# B&R Automation Studio project Fertigungsband
Automation Studio 4.9


## Configuration Kamerainspektion

### Task classes (Cpu.sw)
```
Cyclic#4:
  Verpressen <- Verpressen.prg
```


## Configuration Pressen

CPU X20CP1584, AutomationRuntime J4.93, Build 4.1.2, Vc V4.73.2

### Task classes (Cpu.sw)
```
Cyclic#4:
  Verpressen <- Verpressen.prg
Binaries: udbdef, FWRules, TCData, iomap, ashwac, Role, sysconf, arconfig, asfw, User, asiol2, ashwd
```

### Hardware
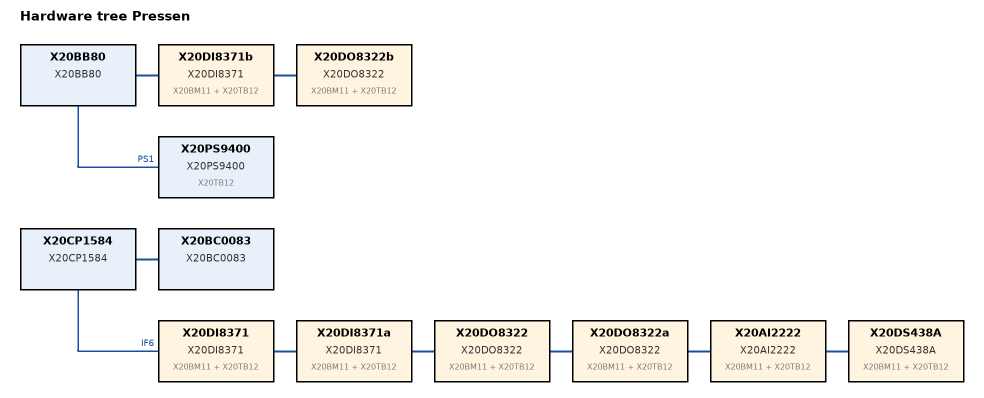
```
X20AI2222 : X20AI2222 v1.2.0.0  [SS1 -> X20TB12d.SS; SL -> X20BM11d.SL1]
X20BB80 : X20BB80 v1.1.0.0
X20BC0083 : X20BC0083 v2.14.0.0  [PLK1 -> X20CP1584.IF3 (NodeNumber=1) [Cable Type=PowerlinkCable, Length=10, Version=1.0.0.3]; SL -> X20BB80.SL1]
X20BM11 : X20BM11 v1.1.0.0  [X2X1 -> X20CP1584.IF6]
X20BM11a : X20BM11 v1.1.0.0  [X2X1 -> X20BM11.X2X2]
X20BM11b : X20BM11 v1.1.0.0  [X2X1 -> X20BM11a.X2X2]
X20BM11c : X20BM11 v1.1.0.0  [X2X1 -> X20BM11b.X2X2]
X20BM11d : X20BM11 v1.1.0.0  [X2X1 -> X20BM11c.X2X2]
X20BM11e : X20BM11 v1.1.0.0  [X2X1 -> X20BM11d.X2X2]
X20BM11f : X20BM11 v1.1.0.0  [X2X1 -> X20BB80.IF1]
X20BM11g : X20BM11 v1.1.0.0  [X2X1 -> X20BM11f.X2X2]
X20CP1584 : X20CP1584 v1.10.0.0
  Connector IF2:
    ActivateDevice = 1
    Mode = Manual
    InternetAddress = 10.36.37.3
    SubnetMask = 255.255.255.0
  ConfigurationID = Fertiungsband_basisConfig
  FileDevice1
  FileDeviceName1 = USER
  FileDevicePath1 = USER_PATH
X20DI8371 : X20DI8371 v1.4.0.0  [SS1 -> X20TB12.SS; SL -> X20BM11.SL1]
X20DI8371a : X20DI8371 v1.4.0.0  [SS1 -> X20TB12a.SS; SL -> X20BM11a.SL1]
X20DI8371b : X20DI8371 v1.4.0.0  [SS1 -> X20TB12g.SS; SL -> X20BM11f.SL1]
X20DO8322 : X20DO8322 v1.5.0.0  [SS1 -> X20TB12b.SS; SL -> X20BM11b.SL1]
X20DO8322a : X20DO8322 v1.5.0.0  [SS1 -> X20TB12c.SS; SL -> X20BM11c.SL1]
X20DO8322b : X20DO8322 v1.5.0.0  [SS1 -> X20TB12h.SS; SL -> X20BM11g.SL1]
X20DS438A : X20DS438A v2.3.0.0  [SS1 -> X20TB12e.SS; SL -> X20BM11e.SL1]
  DtmRef = FBD.BRIOLinkModuleDTM.DTMCore.X20DS438A
  DtmId = 84349467-65e7-4600-9e01-ae0e2285639b
  CommDtmId = 6efde10b-66b8-4cae-87f3-db096a55aaa2
  RequiresDTMBuild = true
  ConfigFile = Communication.dtm
  ConfigModule = asiol2
X20PS9400 : X20PS9400 v1.8.0.0  [SS1 -> X20TB12f.SS; PS -> X20BB80.PS1]
X20TB12 : X20TB12 v1.0.0.0
X20TB12a : X20TB12 v1.0.0.0
X20TB12b : X20TB12 v1.0.0.0
X20TB12c : X20TB12 v1.0.0.0
X20TB12d : X20TB12 v1.0.0.0
X20TB12e : X20TB12 v1.0.0.0
X20TB12f : X20TB12 v1.0.0.0
X20TB12g : X20TB12 v1.0.0.0
X20TB12h : X20TB12 v1.0.0.0
```

### IoMap.iom - X20CP1584/IoMap.iom
```iecst
VAR_CONFIG
	::Werkstueck_Bandende_Links AT %IX."X20DI8371".DigitalInput01;
	::Werkstueck_Bandende_Rechts AT %IX."X20DI8371".DigitalInput02;
	::Koppelsensor_Empfaenger_rechts AT %IX."X20DI8371".DigitalInput03;
	::Koppelsensor_Empfaenger_links AT %IX."X20DI8371".DigitalInput04;
	::Stopper_geoffnet AT %IX."X20DI8371".DigitalInput05;
	::Notaus AT %IX."X20DI8371".DigitalInput06;
	::Motor_Drehgeber1 AT %IX."X20DI8371".DigitalInput07;
	::Motor_Drehgeber2 AT %IX."X20DI8371".DigitalInput08;
	::START_Taster_Gruen AT %IX."X20DI8371a".DigitalInput01;
	::STOP_Taster_Rot AT %IX."X20DI8371a".DigitalInput02;
	::Reset_Taster_Weis AT %IX."X20DI8371a".DigitalInput03;
	::Wahlschalter AT %IX."X20DI8371a".DigitalInput04;
	::AuthCodeBit[0] AT %IX."X20DI8371a".DigitalInput05;
	::AuthCodeBit[1] AT %IX."X20DI8371a".DigitalInput06;
	::AuthCodeBit[2] AT %IX."X20DI8371a".DigitalInput07;
	::AuthCodeBit[3] AT %IX."X20DI8371a".DigitalInput08;
	::Bandantrieb_Rechts AT %QX."X20DO8322".DigitalOutput01;
	::Bandantrieb_Links AT %QX."X20DO8322".DigitalOutput02;
	::Bandantrieb_Schleichgang AT %QX."X20DO8322".DigitalOutput03;
	::Stopper_oeffnen AT %QX."X20DO8322".DigitalOutput04;
	::Koppelsensor_Sender_links AT %QX."X20DO8322".DigitalOutput05;
	::Koppelsensor_Sender_rechts AT %QX."X20DO8322".DigitalOutput06;
	::Lampe_Gruen AT %QX."X20DO8322a".DigitalOutput01;
	::Lampe_Weiss AT %QX."X20DO8322a".DigitalOutput02;
	::Verpressen:Lampe_Q1 AT %QX."X20DO8322a".DigitalOutput03;
	::Verpressen:Lampe_Q2 AT %QX."X20DO8322a".DigitalOutput04;
	::Potentiometer1 AT %IW."X20AI2222".AnalogInput01;
	::Potentiometer2 AT %IW."X20AI2222".AnalogInput02;
	::Verpressen:Zylinder_auf AT %QX."X20DO8322b".DigitalOutput01;
	::Verpressen:Zylinder_ab AT %QX."X20DO8322b".DigitalOutput02;
	::Verpressen:Zylinder_oben AT %IX."X20DI8371b".DigitalInput01;
	::Verpressen:Zylinder_unten AT %IX."X20DI8371b".DigitalInput02;
	::Verpressen:Teil_vorhanden AT %IX."X20DI8371b".DigitalInput08;
END_VAR
```

## Configuration Tunnelofen

### IoMap.iom - X20CP1584/IoMap.iom
```iecst
VAR_CONFIG
	::Werkstueck_Bandende_Links AT %IX."X20DI8371".DigitalInput01;
	::Werkstueck_Bandende_Rechts AT %IX."X20DI8371".DigitalInput02;
	::Koppelsensor_Empfaenger_rechts AT %IX."X20DI8371".DigitalInput03;
	::Koppelsensor_Empfaenger_links AT %IX."X20DI8371".DigitalInput04;
	::Stopper_geoffnet AT %IX."X20DI8371".DigitalInput05;
	::Notaus AT %IX."X20DI8371".DigitalInput06;
	::Motor_Drehgeber1 AT %IX."X20DI8371".DigitalInput07;
	 ::Motor_Drehgeber2 AT %IX."X20DI8371".DigitalInput08;
	::START_Taster_Gruen AT %IX."X20DI8371a".DigitalInput01;
	::STOP_Taster_Rot AT %IX."X20DI8371a".DigitalInput02;
	::Reset_Taster_Weis AT %IX."X20DI8371a".DigitalInput03;
	::Wahlschalter AT %IX."X20DI8371a".DigitalInput04;
	::AuthCodeBit[0] AT %IX."X20DI8371a".DigitalInput05;
	::AuthCodeBit[1] AT %IX."X20DI8371a".DigitalInput06;
	::AuthCodeBit[2]  AT %IX."X20DI8371a".DigitalInput07;
	::AuthCodeBit[3]  AT %IX."X20DI8371a".DigitalInput08;
	::Bandantrieb_Rechts AT %QX."X20DO8322".DigitalOutput01;
	::Bandantrieb_Links AT %QX."X20DO8322".DigitalOutput02;
	::Bandantrieb_Schleichgang AT %QX."X20DO8322".DigitalOutput03;
	::Stopper_oeffnen AT %QX."X20DO8322".DigitalOutput04;
	::Koppelsensor_Sender_links AT %QX."X20DO8322".DigitalOutput05;
	::Koppelsensor_Sender_rechts AT %QX."X20DO8322".DigitalOutput06;
	::Lampe_Gruen AT %QX."X20DO8322a".DigitalOutput01;
	::Lampe_Weiss AT %QX."X20DO8322a".DigitalOutput02;
	::Lampe_Q1_Weiss AT %QX."X20DO8322a".DigitalOutput03;
	::Lampe_Q2_Weiss AT %QX."X20DO8322a".DigitalOutput04;
	::Potentiometer1 AT %IW."X20AI2222".AnalogInput01;
	::Potentiometer2 AT %IW."X20AI2222".AnalogInput02;
END_VAR
```

## Configuration Wenden

CPU X20CP1584, AutomationRuntime J4.93, Build 4.1.2, Vc V4.73.2

### Hardware
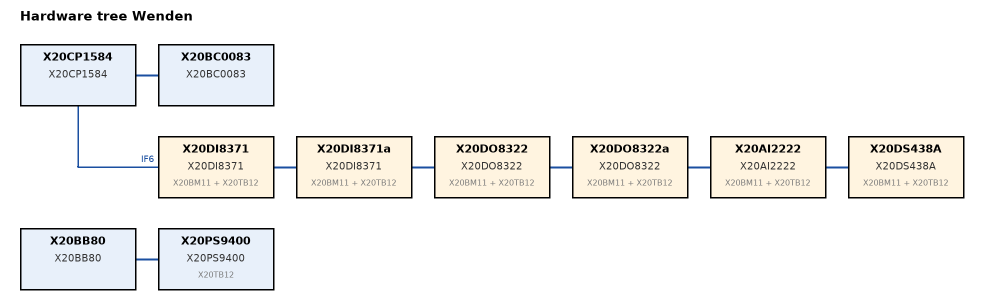
```
X20AI2222 : X20AI2222 v1.2.0.0  [SS1 -> X20TB12d.SS; SL -> X20BM11d.SL1]
X20BB80 : X20BB80 v1.1.0.0
X20BC0083 : X20BC0083 v2.14.0.0  [PLK1 -> X20CP1584.IF3 (NodeNumber=1) [Cable Type=PowerlinkCable, Length=10, Version=1.0.0.3]; SL -> X20BB80.SL1]
X20BM11 : X20BM11 v1.1.0.0  [X2X1 -> X20CP1584.IF6]
X20BM11a : X20BM11 v1.1.0.0  [X2X1 -> X20BM11.X2X2]
X20BM11b : X20BM11 v1.1.0.0  [X2X1 -> X20BM11a.X2X2]
X20BM11c : X20BM11 v1.1.0.0  [X2X1 -> X20BM11b.X2X2]
X20BM11d : X20BM11 v1.1.0.0  [X2X1 -> X20BM11c.X2X2]
X20BM11e : X20BM11 v1.1.0.0  [X2X1 -> X20BM11d.X2X2]
X20CP1584 : X20CP1584 v1.10.0.0
  Connector IF2:
    ActivateDevice = 1
  ConfigurationID = Fertiungsband_basisConfig
  FileDevice1
  FileDeviceName1 = USER
  FileDevicePath1 = USER_PATH
X20DI8371 : X20DI8371 v1.4.0.0  [SS1 -> X20TB12.SS; SL -> X20BM11.SL1]
X20DI8371a : X20DI8371 v1.4.0.0  [SS1 -> X20TB12a.SS; SL -> X20BM11a.SL1]
X20DO8322 : X20DO8322 v1.5.0.0  [SS1 -> X20TB12b.SS; SL -> X20BM11b.SL1]
X20DO8322a : X20DO8322 v1.5.0.0  [SS1 -> X20TB12c.SS; SL -> X20BM11c.SL1]
X20DS438A : X20DS438A v2.3.0.0  [SS1 -> X20TB12e.SS; SL -> X20BM11e.SL1]
  DtmRef = FBD.BRIOLinkModuleDTM.DTMCore.X20DS438A
  DtmId = 84349467-65e7-4600-9e01-ae0e2285639b
  CommDtmId = 6efde10b-66b8-4cae-87f3-db096a55aaa2
  RequiresDTMBuild = true
  ConfigFile = Communication.dtm
  ConfigModule = asiol2
X20PS9400 : X20PS9400 v1.8.0.0  [SS1 -> X20TB12f.SS; PS -> X20BB80.PS1]
X20TB12 : X20TB12 v1.0.0.0
X20TB12a : X20TB12 v1.0.0.0
X20TB12b : X20TB12 v1.0.0.0
X20TB12c : X20TB12 v1.0.0.0
X20TB12d : X20TB12 v1.0.0.0
X20TB12e : X20TB12 v1.0.0.0
X20TB12f : X20TB12 v1.0.0.0
```

## Logical view

### Global.var - Global variables
```iecst
VAR
	Werkstueck_Bandende_Links 		: BOOL;
	Werkstueck_Bandende_Rechts 		: BOOL;
	Koppelsensor_Empfaenger_rechts 	: BOOL;
	Koppelsensor_Empfaenger_links 	: BOOL;
	Stopper_geoffnet 				: BOOL;
	Notaus 							: BOOL;
	Motor_Drehgeber1 				: BOOL;
	Motor_Drehgeber2 				: BOOL;
	START_Taster_Gruen 				: BOOL;
	STOP_Taster_Rot					: BOOL;
	Reset_Taster_Weis 				: BOOL;
	Wahlschalter 					: BOOL;
	AuthCodeBit 					: ARRAY[0..3] OF BOOL;
	Bandantrieb_Rechts				: BOOL;
	Bandantrieb_Links				: BOOL;
	Bandantrieb_Schleichgang		: BOOL;
	Stopper_oeffnen					: BOOL;
	Koppelsensor_Sender_links		: BOOL;
	Koppelsensor_Sender_rechts		: BOOL;
	Lampe_Gruen						: BOOL;
	Lampe_Weiss						: BOOL;
	Lampe_Q1_Weiss					: BOOL;
	Lampe_Q2_Weiss					: BOOL;
	Potentiometer1					: INT;
	Potentiometer2					: INT;
	RFID_Reader						: STRING;
END_VAR
```

### Verpressen.var
```iecst
VAR
	Zylinder_oben : BOOL;
	Zylinder_unten : BOOL;
	Zylinder_auf : BOOL;
	Zylinder_ab : BOOL;
	Teil_vorhanden : BOOL;
END_VAR
```

### Program Logical/Verpressen (ANSIC)

#### Types.typ
```iecst
TYPE
	Status_t :
		(
		INIT,
		BEREIT,
		ZYLINDER_AB,
		ZYLINDER_AUF,
		FERTIG,
		FEHLER
		);
END_TYPE
```

#### Variables.var
```iecst
VAR
	Zylinder_oben : BOOL;
	Zylinder_unten : BOOL;
	Zylinder_auf : BOOL;
	Zylinder_ab : BOOL;
	Teil_vorhanden : BOOL;
	Status : Status_t;
	Lampe_Q1 : BOOL;
	Lampe_Q2 : BOOL;
END_VAR
```

#### Cyclic.c
```c
#include <bur/plctypes.h>

#ifdef _DEFAULT_INCLUDES
	#include <AsDefault.h>
#endif

void _CYCLIC ProgramCyclic(void)
{
	// TODO Error Handling

	switch (Status)
	{
		case INIT:
			if (Zylinder_oben)
			{
				Zylinder_auf = 0;
				Status = BEREIT;
			}
			break;

		case BEREIT:
			if (Teil_vorhanden)
			{
				Lampe_Q2 = 1;
				Zylinder_ab = 1;
				Status = ZYLINDER_AB;
			}
			break;

		case ZYLINDER_AB:
			if (Zylinder_unten)
			{
				Zylinder_ab = 0;
				Zylinder_auf = 1;
				Status = ZYLINDER_AUF;
			}
			break;

		case ZYLINDER_AUF:
			if (Zylinder_oben)
			{
				Zylinder_auf = 0;
				Lampe_Q2 = 0;
				Status = FERTIG;
			}
			break;

		case FERTIG:
			if (!Teil_vorhanden)
			{
				Status = BEREIT;
			}
			break;

		case FEHLER:
			// TODO
			Zylinder_auf = 0;
			Zylinder_ab = 0;
			Lampe_Q1 = 1;
			Lampe_Q2 = 0;
			break;

		default:
			Status = FEHLER;
			break;
	}
}
```

#### Init.c
```c
#include <bur/plctypes.h>

#ifdef _DEFAULT_INCLUDES
	#include <AsDefault.h>
#endif

void _INIT ProgramInit(void)
{
	Lampe_Q2 = 0;

	if (Zylinder_oben)
	{
		Zylinder_auf = 0;
		Zylinder_ab = 0;
		Status = BEREIT;
	}
	else
	{
		Zylinder_auf = 1;
		Zylinder_ab = 0;
		Status = INIT;
	}
}
```

Listed in the project but not available here: Logical/Global.typ, Logical/Libraries
